TYPE TMethodNames_Cohap :
STRUCT
	M_init : STRING := 'init';
	M_GetAsicandChannelCardVersion : STRING := 'getSICAndChannelCardVersions';
	M_GetDLLVersion : STRING := 'getDLLVersions';
	M_TestDummy : STRING := 'TestDummy';
	M_TestDummy2 : STRING := 'TestDummy2';
	M_PowerUp : STRING := 'PowerUp';
	M_PowerDown : STRING := 'PowerDown';
	M_readSerialNumber : STRING := 'readSerialNumber';
	M_ReadDeviceOutput : STRING := 'ReadDeviceOutput';
	M_ReadFastChannelData : STRING := 'SENT_readFastChannelData';
	M_initDUT : STRING := 'initDUT';
	M_initialize : STRING := 'initialize';
	
	M_InitLot : STRING := 'InitLot';
END_STRUCT
END_TYPE

(* stored: Version 1.1.0.1, ProductVersion 3.1.4024.12
   DUT TMethodNames_Cohap: Id {b95cf753-0d18-4208-847a-8e335e6d67c0} *)
